% RSLogix 500 project Unscrambler_D.RSS, saved by version 12.00.00.00 %
PROJECT "3234"    % processor: MicroLogix 1400 %

PROGRAM FILES
  LAD 2   15 rungs
  LAD 3   13 rungs
  LAD 4   2 rungs
  LAD 5   18 rungs
  LAD 6   37 rungs
  LAD 7   31 rungs
  LAD 8   105 rungs
  LAD 9, 10, 11, 12, 13, 14, 15: only END

DATA FILES
  O0 OUTPUT  6 elements
  I1 INPUT  9 elements
  S2 STATUS  66 elements
  B3 BINARY  32 elements
  T4 TIMER  40 elements
  C5 COUNTER  32 elements
  R6 CONTROL  16 elements
  N7 INTEGER  105 elements
  F8 FLOAT  1 elements
  N10   10 elements
  MG11   40 elements
  N12   2 elements
  N13   10 elements
  N17   1 elements
  ST23   32 elements
  N24   17 elements
  B27   1 elements

LADDER 2
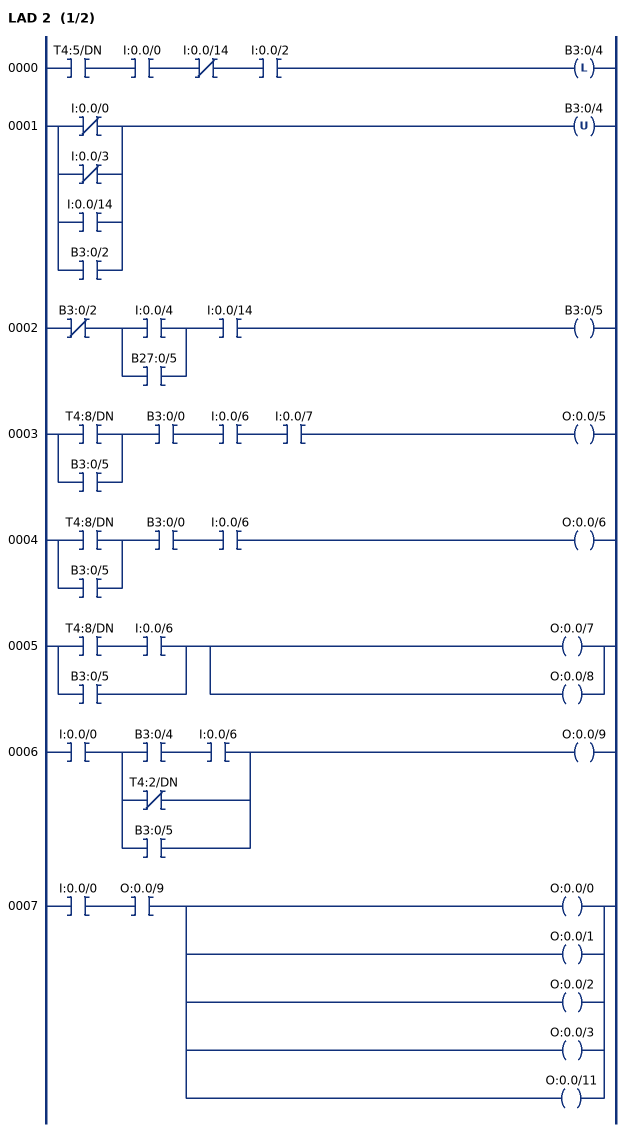
% Rung: 0 %
SOR XIC T4:5/DN XIC I:0.0/0 XIO I:0.0/14 XIC I:0.0/2 OTL B3:0/4 EOR
% Rung: 1 %
SOR BST XIO I:0.0/0 NXB XIO I:0.0/3 NXB XIC I:0.0/14 NXB XIC B3:0/2 BND OTU B3:0/4 EOR
% Rung: 2 %
SOR XIO B3:0/2 BST XIC I:0.0/4 NXB XIC B27:0/5 BND XIC I:0.0/14 OTE B3:0/5 EOR
% Rung: 3 %
SOR BST XIC T4:8/DN NXB XIC B3:0/5 BND XIC B3:0/0 XIC I:0.0/6 XIC I:0.0/7 OTE O:0.0/5 EOR
% Rung: 4 %
SOR BST XIC T4:8/DN NXB XIC B3:0/5 BND XIC B3:0/0 XIC I:0.0/6 OTE O:0.0/6 EOR
% Rung: 5 %
SOR BST XIC T4:8/DN XIC I:0.0/6 NXB XIC B3:0/5 BND BST OTE O:0.0/7 NXB OTE O:0.0/8 BND EOR
% Rung: 6 %
SOR XIC I:0.0/0 BST XIC B3:0/4 XIC I:0.0/6 NXB XIO T4:2/DN NXB XIC B3:0/5 BND OTE O:0.0/9 EOR
% Rung: 7 %
SOR XIC I:0.0/0 XIC O:0.0/9 BST OTE O:0.0/0 NXB OTE O:0.0/1 NXB OTE O:0.0/2 NXB OTE O:0.0/3 NXB OTE O:0.0/11 BND EOR

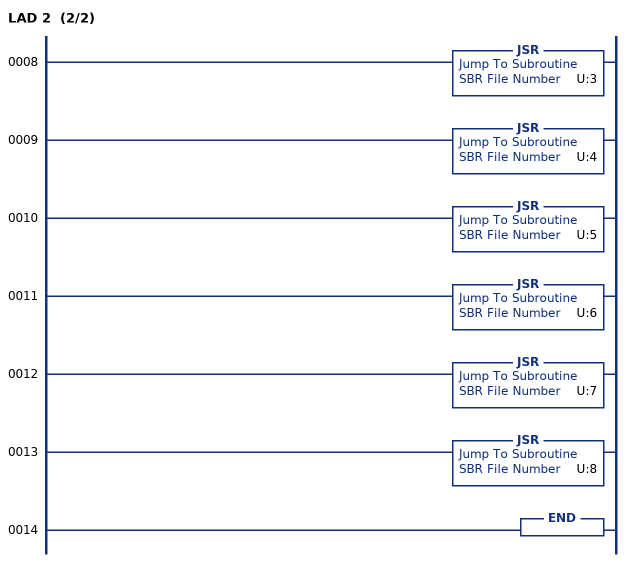
% Rung: 8 %
SOR JSR U:3 EOR
% Rung: 9 %
SOR JSR U:4 EOR
% Rung: 10 %
SOR JSR U:5 EOR
% Rung: 11 %
SOR JSR U:6 EOR
% Rung: 12 %
SOR JSR U:7 EOR
% Rung: 13 %
SOR JSR U:8 EOR
% Rung: 14 %
SOR END EOR

LADDER 3
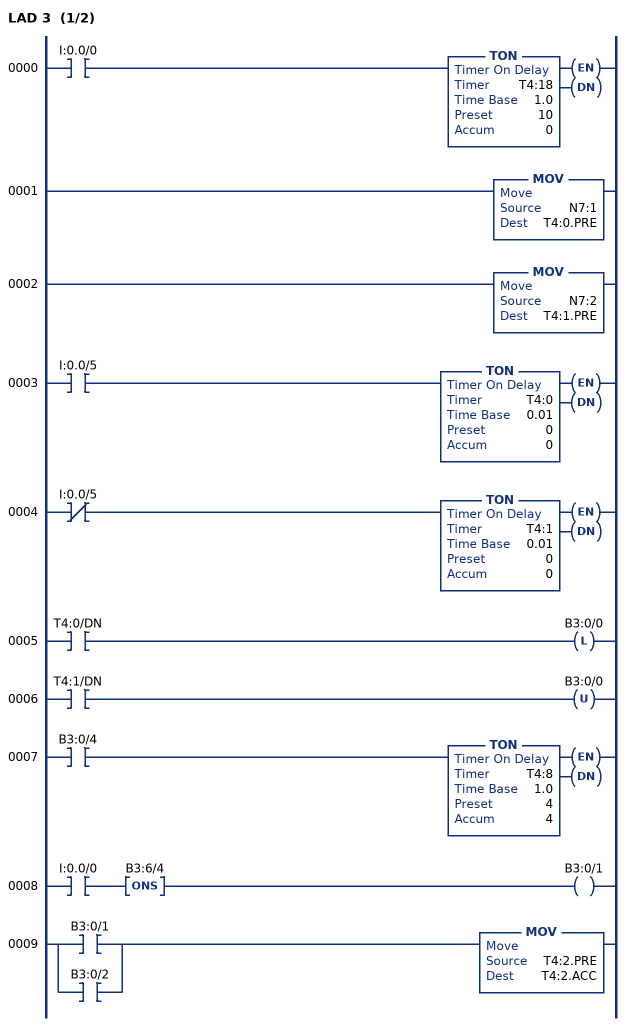
% Rung: 0 %
SOR XIC I:0.0/0 TON T4:18 1.0 10 0 EOR
% Rung: 1 %
SOR MOV N7:1 T4:0.PRE EOR
% Rung: 2 %
SOR MOV N7:2 T4:1.PRE EOR
% Rung: 3 %
SOR XIC I:0.0/5 TON T4:0 0.01 0 0 EOR
% Rung: 4 %
SOR XIO I:0.0/5 TON T4:1 0.01 0 0 EOR
% Rung: 5 %
SOR XIC T4:0/DN OTL B3:0/0 EOR
% Rung: 6 %
SOR XIC T4:1/DN OTU B3:0/0 EOR
% Rung: 7 %
SOR XIC B3:0/4 TON T4:8 1.0 4 4 EOR
% Rung: 8 %
SOR XIC I:0.0/0 ONS B3:6/4 OTE B3:0/1 EOR
% Rung: 9 %
SOR BST XIC B3:0/1 NXB XIC B3:0/2 BND MOV T4:2.PRE T4:2.ACC EOR

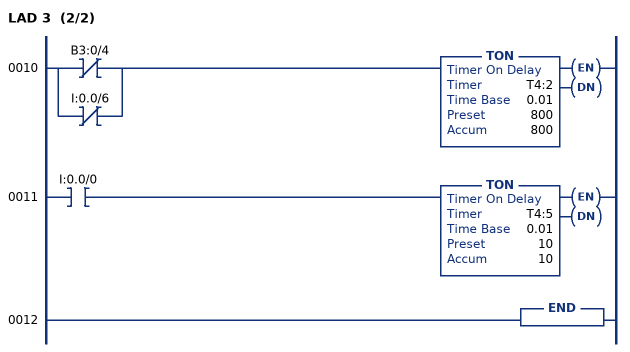
% Rung: 10 %
SOR BST XIO B3:0/4 NXB XIO I:0.0/6 BND TON T4:2 0.01 800 800 EOR
% Rung: 11 %
SOR XIC I:0.0/0 TON T4:5 0.01 10 10 EOR
% Rung: 12 %
SOR END EOR

LADDER 4
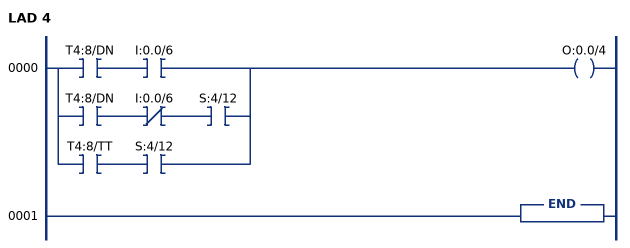
% Rung: 0 %
SOR BST XIC T4:8/DN XIC I:0.0/6 NXB XIC T4:8/DN XIO I:0.0/6 XIC S:4/12 NXB XIC T4:8/TT XIC S:4/12 BND OTE O:0.0/4 EOR
% Rung: 1 %
SOR END EOR

LADDER 5
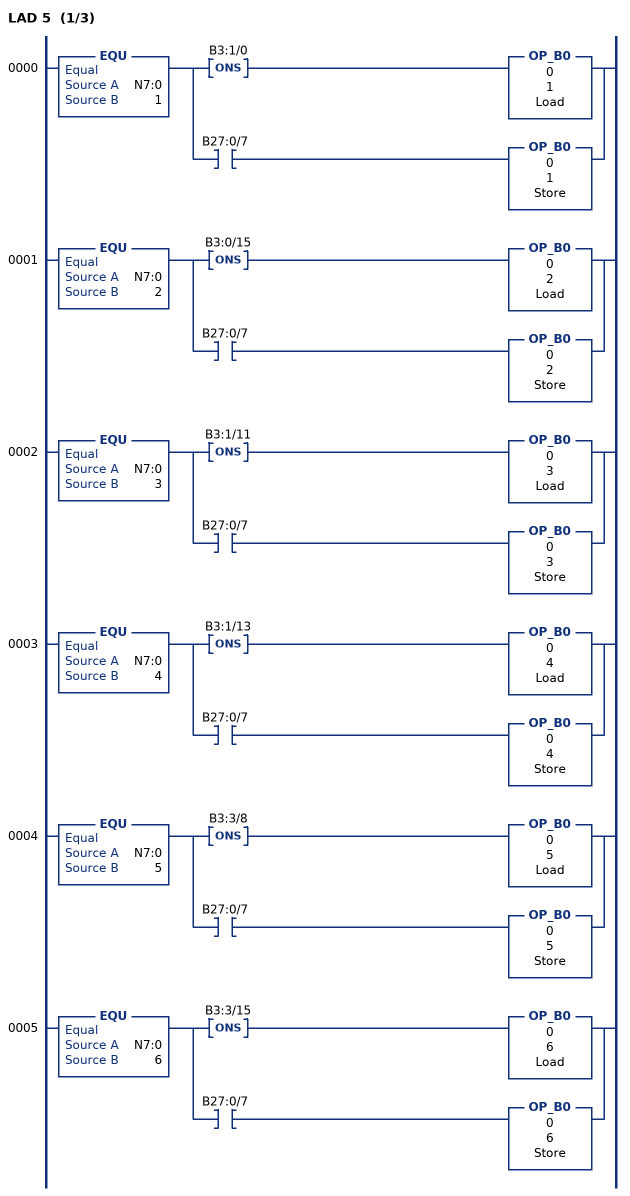
% Rung: 0 %
SOR EQU N7:0 1 BST ONS B3:1/0 OP_B0 0 1 Load NXB XIC B27:0/7 OP_B0 0 1 Store BND EOR
% Rung: 1 %
SOR EQU N7:0 2 BST ONS B3:0/15 OP_B0 0 2 Load NXB XIC B27:0/7 OP_B0 0 2 Store BND EOR
% Rung: 2 %
SOR EQU N7:0 3 BST ONS B3:1/11 OP_B0 0 3 Load NXB XIC B27:0/7 OP_B0 0 3 Store BND EOR
% Rung: 3 %
SOR EQU N7:0 4 BST ONS B3:1/13 OP_B0 0 4 Load NXB XIC B27:0/7 OP_B0 0 4 Store BND EOR
% Rung: 4 %
SOR EQU N7:0 5 BST ONS B3:3/8 OP_B0 0 5 Load NXB XIC B27:0/7 OP_B0 0 5 Store BND EOR
% Rung: 5 %
SOR EQU N7:0 6 BST ONS B3:3/15 OP_B0 0 6 Load NXB XIC B27:0/7 OP_B0 0 6 Store BND EOR

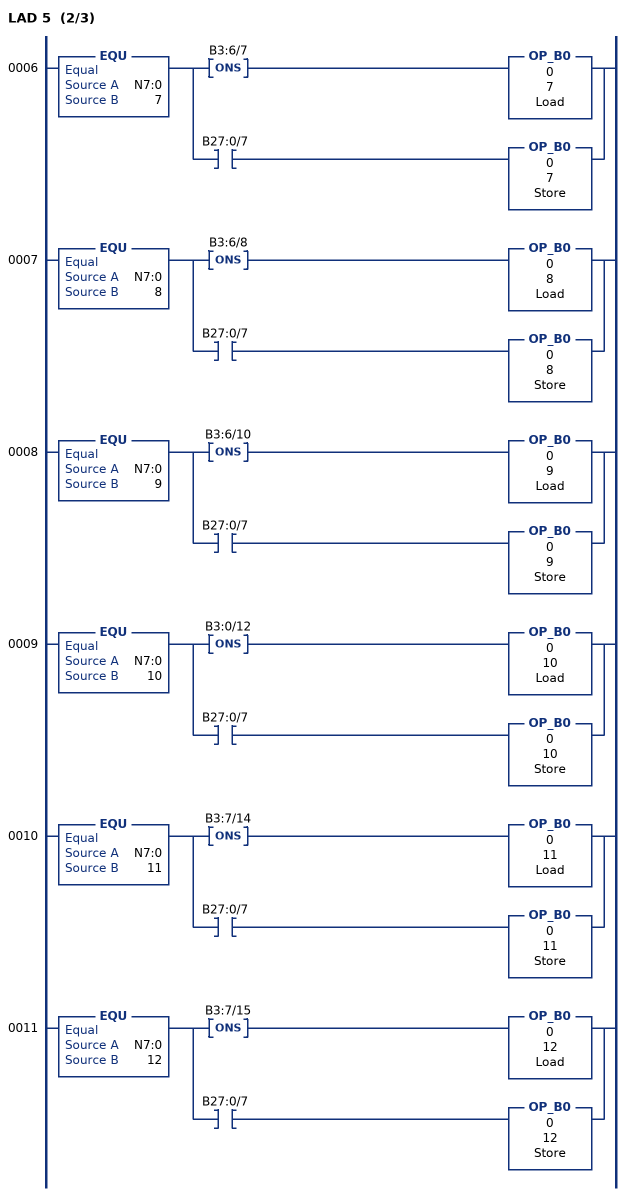
% Rung: 6 %
SOR EQU N7:0 7 BST ONS B3:6/7 OP_B0 0 7 Load NXB XIC B27:0/7 OP_B0 0 7 Store BND EOR
% Rung: 7 %
SOR EQU N7:0 8 BST ONS B3:6/8 OP_B0 0 8 Load NXB XIC B27:0/7 OP_B0 0 8 Store BND EOR
% Rung: 8 %
SOR EQU N7:0 9 BST ONS B3:6/10 OP_B0 0 9 Load NXB XIC B27:0/7 OP_B0 0 9 Store BND EOR
% Rung: 9 %
SOR EQU N7:0 10 BST ONS B3:0/12 OP_B0 0 10 Load NXB XIC B27:0/7 OP_B0 0 10 Store BND EOR
% Rung: 10 %
SOR EQU N7:0 11 BST ONS B3:7/14 OP_B0 0 11 Load NXB XIC B27:0/7 OP_B0 0 11 Store BND EOR
% Rung: 11 %
SOR EQU N7:0 12 BST ONS B3:7/15 OP_B0 0 12 Load NXB XIC B27:0/7 OP_B0 0 12 Store BND EOR

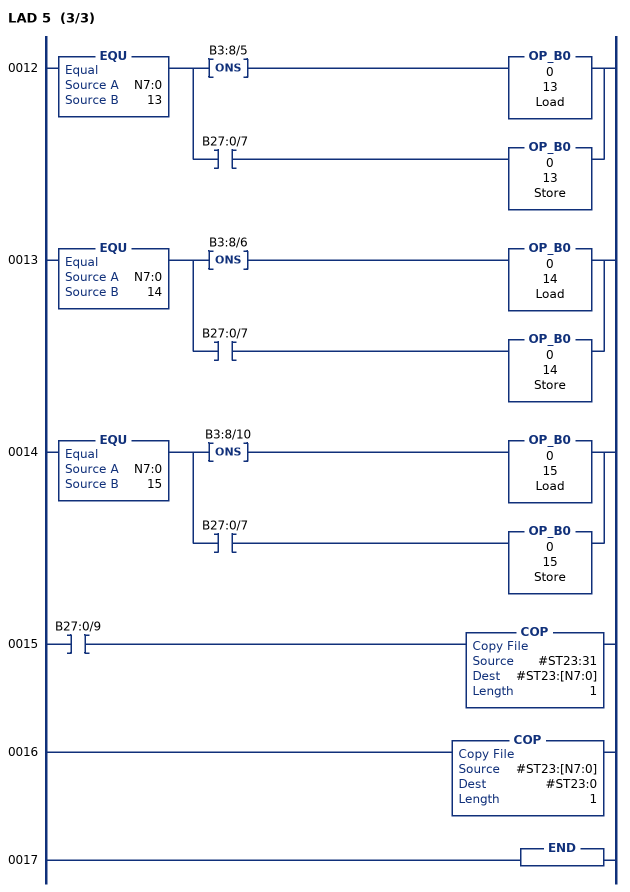
% Rung: 12 %
SOR EQU N7:0 13 BST ONS B3:8/5 OP_B0 0 13 Load NXB XIC B27:0/7 OP_B0 0 13 Store BND EOR
% Rung: 13 %
SOR EQU N7:0 14 BST ONS B3:8/6 OP_B0 0 14 Load NXB XIC B27:0/7 OP_B0 0 14 Store BND EOR
% Rung: 14 %
SOR EQU N7:0 15 BST ONS B3:8/10 OP_B0 0 15 Load NXB XIC B27:0/7 OP_B0 0 15 Store BND EOR
% Rung: 15 %
SOR XIC B27:0/9 COP #ST23:31 #ST23:[N7:0] 1 EOR
% Rung: 16 %
SOR COP #ST23:[N7:0] #ST23:0 1 EOR
% Rung: 17 %
SOR END EOR

LADDER 6
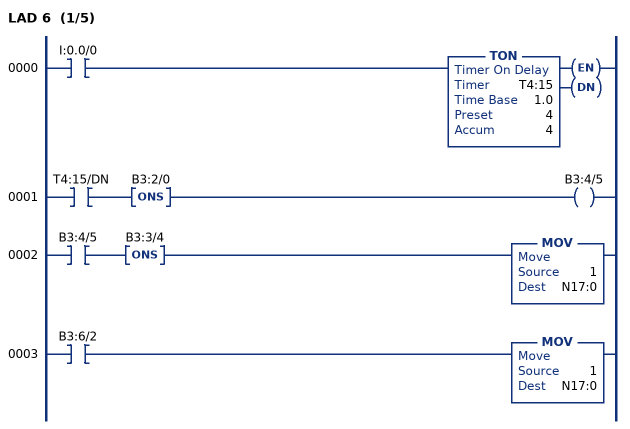
% Rung: 0 %
SOR XIC I:0.0/0 TON T4:15 1.0 4 4 EOR
% Rung: 1 %
SOR XIC T4:15/DN ONS B3:2/0 OTE B3:4/5 EOR
% Rung: 2 %
SOR XIC B3:4/5 ONS B3:3/4 MOV 1 N17:0 EOR
% Rung: 3 %
SOR XIC B3:6/2 MOV 1 N17:0 EOR

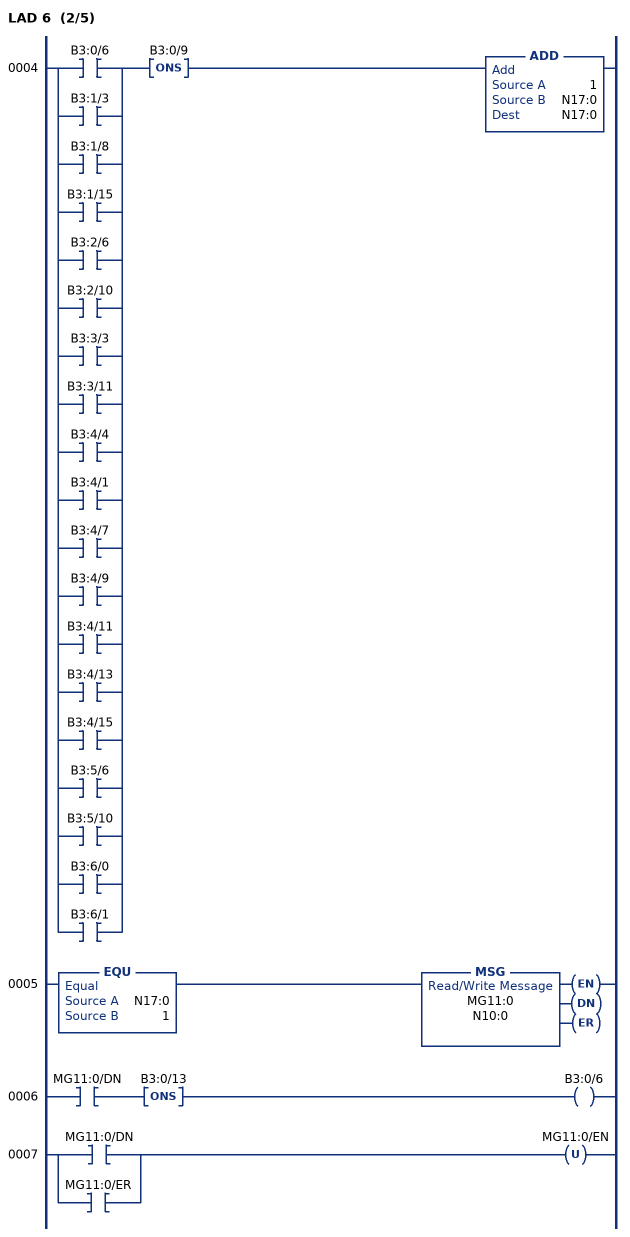
% Rung: 4 %
SOR BST XIC B3:0/6 NXB XIC B3:1/3 NXB XIC B3:1/8 NXB XIC B3:1/15 NXB XIC B3:2/6 NXB XIC B3:2/10 NXB XIC B3:3/3 NXB XIC B3:3/11 NXB XIC B3:4/4 NXB XIC B3:4/1 NXB XIC B3:4/7 NXB XIC B3:4/9 NXB XIC B3:4/11 NXB XIC B3:4/13 NXB XIC B3:4/15 NXB XIC B3:5/6 NXB XIC B3:5/10 NXB XIC B3:6/0 NXB XIC B3:6/1 BND ONS B3:0/9 ADD 1 N17:0 N17:0 EOR
% Rung: 5 %
SOR EQU N17:0 1 MSG MG11:0 N10:0 EOR
%   MSG set-up: 06 Write Single Register (4xxxxx) | 2 | 1 | 8194 | N10:0 | 0 | 1 | 0 | CLIENT              :502 | 0 | 0 | ? %
% Rung: 6 %
SOR XIC MG11:0/DN ONS B3:0/13 OTE B3:0/6 EOR
% Rung: 7 %
SOR BST XIC MG11:0/DN NXB XIC MG11:0/ER BND OTU MG11:0/EN EOR

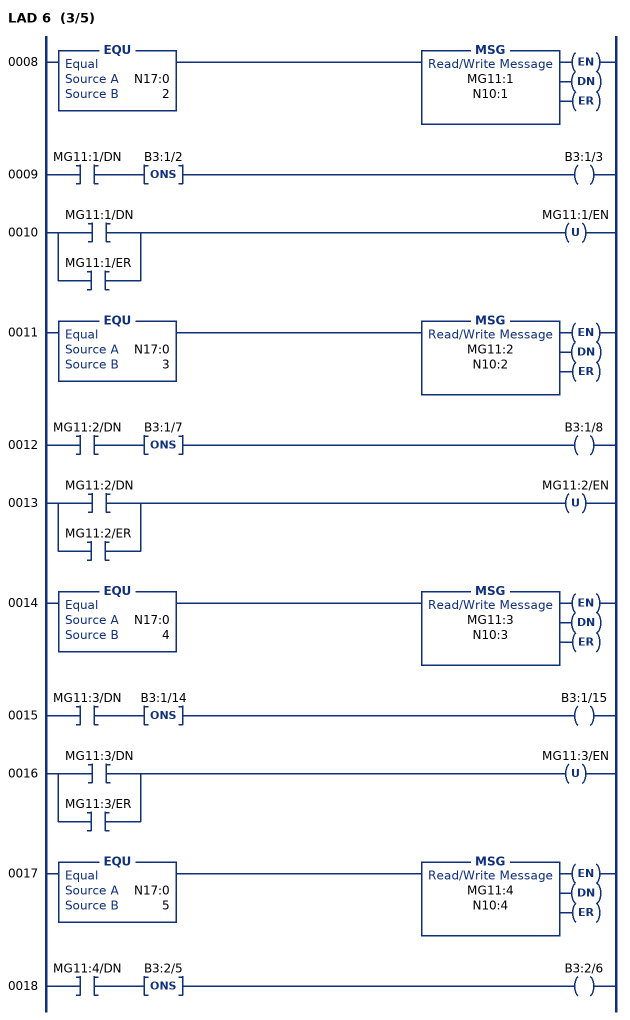
% Rung: 8 %
SOR EQU N17:0 2 MSG MG11:1 N10:1 EOR
%   MSG set-up: 06 Write Single Register (4xxxxx) | 2 | 1 | 8194 | N10:1 | 0 | 2 | 0 | CLIENT              :502 | 0 | 0 | ? %
% Rung: 9 %
SOR XIC MG11:1/DN ONS B3:1/2 OTE B3:1/3 EOR
% Rung: 10 %
SOR BST XIC MG11:1/DN NXB XIC MG11:1/ER BND OTU MG11:1/EN EOR
% Rung: 11 %
SOR EQU N17:0 3 MSG MG11:2 N10:2 EOR
%   MSG set-up: 06 Write Single Register (4xxxxx) | 2 | 1 | 8194 | N10:2 | 0 | 3 | 0 | CLIENT              :502 | 0 | 0 | ? %
% Rung: 12 %
SOR XIC MG11:2/DN ONS B3:1/7 OTE B3:1/8 EOR
% Rung: 13 %
SOR BST XIC MG11:2/DN NXB XIC MG11:2/ER BND OTU MG11:2/EN EOR
% Rung: 14 %
SOR EQU N17:0 4 MSG MG11:3 N10:3 EOR
%   MSG set-up: 06 Write Single Register (4xxxxx) | 2 | 1 | 8194 | N10:3 | 0 | 4 | 0 | CLIENT              :502 | 0 | 0 | ? %
% Rung: 15 %
SOR XIC MG11:3/DN ONS B3:1/14 OTE B3:1/15 EOR
% Rung: 16 %
SOR BST XIC MG11:3/DN NXB XIC MG11:3/ER BND OTU MG11:3/EN EOR
% Rung: 17 %
SOR EQU N17:0 5 MSG MG11:4 N10:4 EOR
%   MSG set-up: 06 Write Single Register (4xxxxx) | 2 | 1 | 8194 | N10:4 | 0 | 5 | 0 | CLIENT              :502 | 0 | 0 | ? %
% Rung: 18 %
SOR XIC MG11:4/DN ONS B3:2/5 OTE B3:2/6 EOR

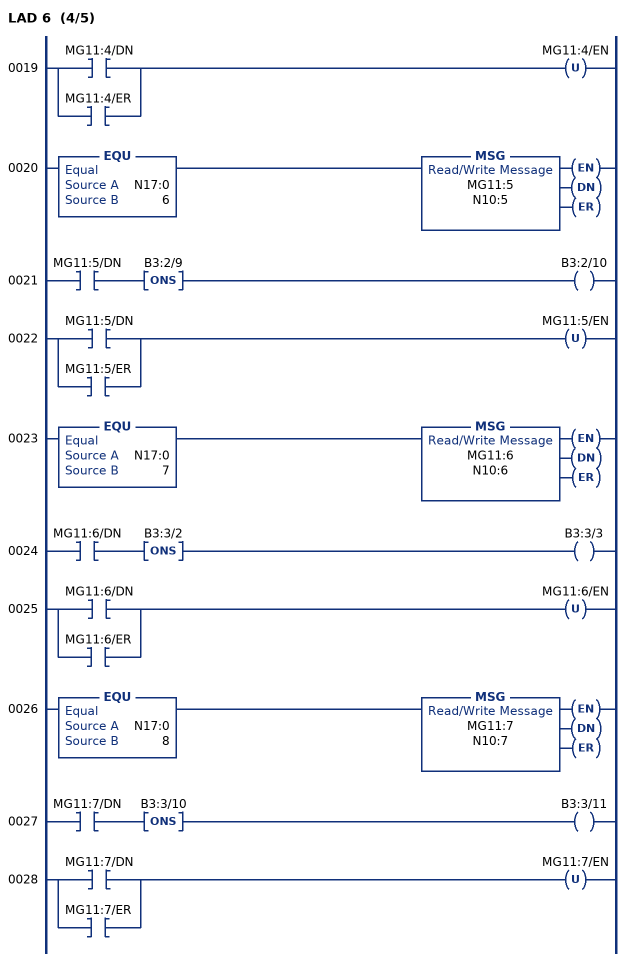
% Rung: 19 %
SOR BST XIC MG11:4/DN NXB XIC MG11:4/ER BND OTU MG11:4/EN EOR
% Rung: 20 %
SOR EQU N17:0 6 MSG MG11:5 N10:5 EOR
%   MSG set-up: 06 Write Single Register (4xxxxx) | 2 | 1 | 8194 | N10:5 | 0 | 6 | 0 | CLIENT              :502 | 0 | 0 | ? %
% Rung: 21 %
SOR XIC MG11:5/DN ONS B3:2/9 OTE B3:2/10 EOR
% Rung: 22 %
SOR BST XIC MG11:5/DN NXB XIC MG11:5/ER BND OTU MG11:5/EN EOR
% Rung: 23 %
SOR EQU N17:0 7 MSG MG11:6 N10:6 EOR
%   MSG set-up: 06 Write Single Register (4xxxxx) | 2 | 1 | 8194 | N10:6 | 0 | 7 | 0 | CLIENT              :502 | 0 | 0 | ? %
% Rung: 24 %
SOR XIC MG11:6/DN ONS B3:3/2 OTE B3:3/3 EOR
% Rung: 25 %
SOR BST XIC MG11:6/DN NXB XIC MG11:6/ER BND OTU MG11:6/EN EOR
% Rung: 26 %
SOR EQU N17:0 8 MSG MG11:7 N10:7 EOR
%   MSG set-up: 06 Write Single Register (4xxxxx) | 2 | 1 | 8194 | N10:7 | 0 | 8 | 0 | CLIENT              :502 | 0 | 0 | ? %
% Rung: 27 %
SOR XIC MG11:7/DN ONS B3:3/10 OTE B3:3/11 EOR
% Rung: 28 %
SOR BST XIC MG11:7/DN NXB XIC MG11:7/ER BND OTU MG11:7/EN EOR

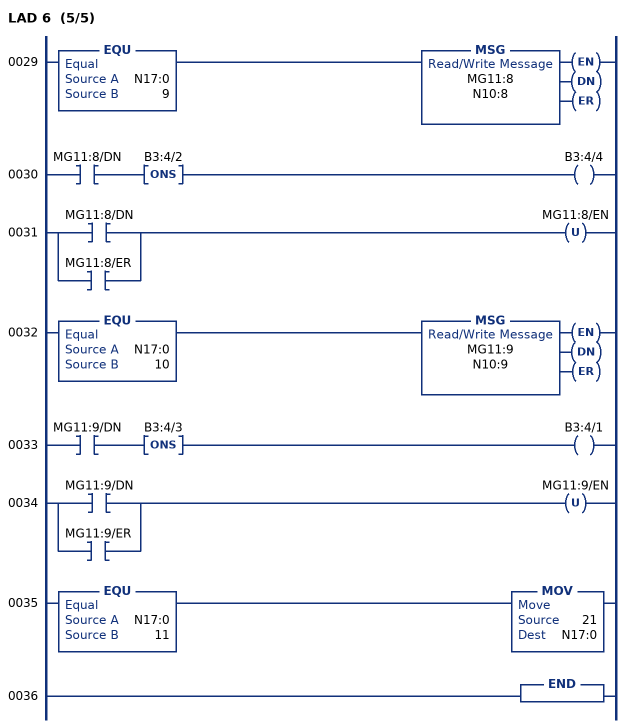
% Rung: 29 %
SOR EQU N17:0 9 MSG MG11:8 N10:8 EOR
%   MSG set-up: 06 Write Single Register (4xxxxx) | 2 | 1 | 8194 | N10:8 | 0 | 9 | 0 | CLIENT              :502 | 0 | 0 | ? %
% Rung: 30 %
SOR XIC MG11:8/DN ONS B3:4/2 OTE B3:4/4 EOR
% Rung: 31 %
SOR BST XIC MG11:8/DN NXB XIC MG11:8/ER BND OTU MG11:8/EN EOR
% Rung: 32 %
SOR EQU N17:0 10 MSG MG11:9 N10:9 EOR
%   MSG set-up: 06 Write Single Register (4xxxxx) | 2 | 1 | 8194 | N10:9 | 0 | 10 | 0 | CLIENT              :502 | 0 | 0 | ? %
% Rung: 33 %
SOR XIC MG11:9/DN ONS B3:4/3 OTE B3:4/1 EOR
% Rung: 34 %
SOR BST XIC MG11:9/DN NXB XIC MG11:9/ER BND OTU MG11:9/EN EOR
% Rung: 35 %
SOR EQU N17:0 11 MOV 21 N17:0 EOR
% Rung: 36 %
SOR END EOR

LADDER 7
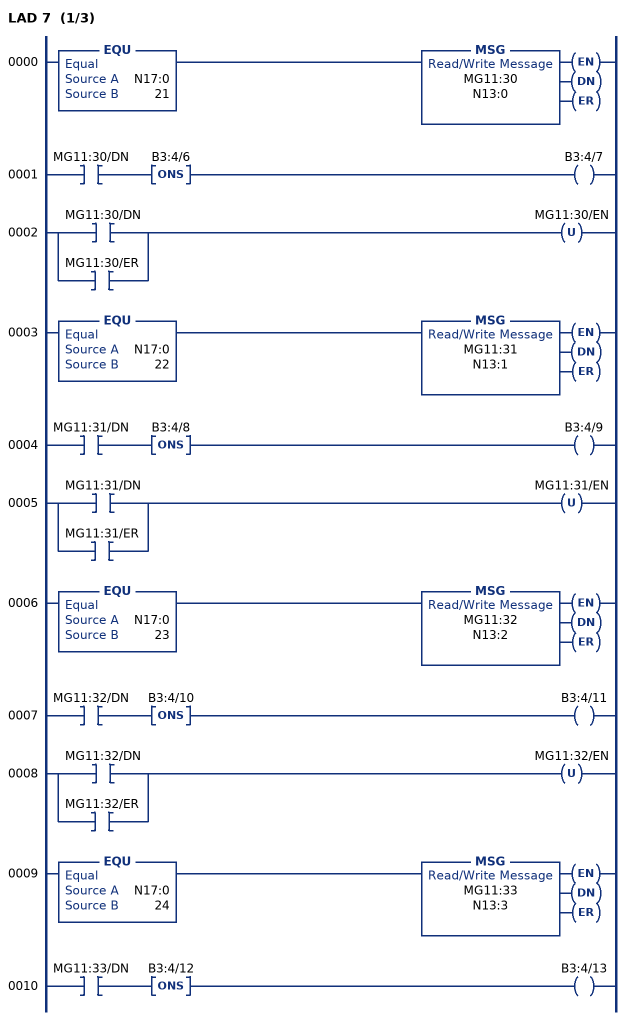
% Rung: 0 %
SOR EQU N17:0 21 MSG MG11:30 N13:0 EOR
%   MSG set-up: 03 Read Holding Registers (4xxxxx) | 5 | 1 | 8449 | N13:0 | 0 | 1 | 0 | CLIENT              :502 | 0 | 0 | ? %
% Rung: 1 %
SOR XIC MG11:30/DN ONS B3:4/6 OTE B3:4/7 EOR
% Rung: 2 %
SOR BST XIC MG11:30/DN NXB XIC MG11:30/ER BND OTU MG11:30/EN EOR
% Rung: 3 %
SOR EQU N17:0 22 MSG MG11:31 N13:1 EOR
%   MSG set-up: 03 Read Holding Registers (4xxxxx) | 5 | 1 | 8449 | N13:1 | 0 | 2 | 0 | CLIENT              :502 | 0 | 0 | ? %
% Rung: 4 %
SOR XIC MG11:31/DN ONS B3:4/8 OTE B3:4/9 EOR
% Rung: 5 %
SOR BST XIC MG11:31/DN NXB XIC MG11:31/ER BND OTU MG11:31/EN EOR
% Rung: 6 %
SOR EQU N17:0 23 MSG MG11:32 N13:2 EOR
%   MSG set-up: 03 Read Holding Registers (4xxxxx) | 5 | 1 | 8449 | N13:2 | 0 | 3 | 0 | CLIENT              :502 | 0 | 0 | ? %
% Rung: 7 %
SOR XIC MG11:32/DN ONS B3:4/10 OTE B3:4/11 EOR
% Rung: 8 %
SOR BST XIC MG11:32/DN NXB XIC MG11:32/ER BND OTU MG11:32/EN EOR
% Rung: 9 %
SOR EQU N17:0 24 MSG MG11:33 N13:3 EOR
%   MSG set-up: 03 Read Holding Registers (4xxxxx) | 5 | 1 | 8449 | N13:3 | 0 | 4 | 0 | CLIENT              :502 | 0 | 0 | ? %
% Rung: 10 %
SOR XIC MG11:33/DN ONS B3:4/12 OTE B3:4/13 EOR

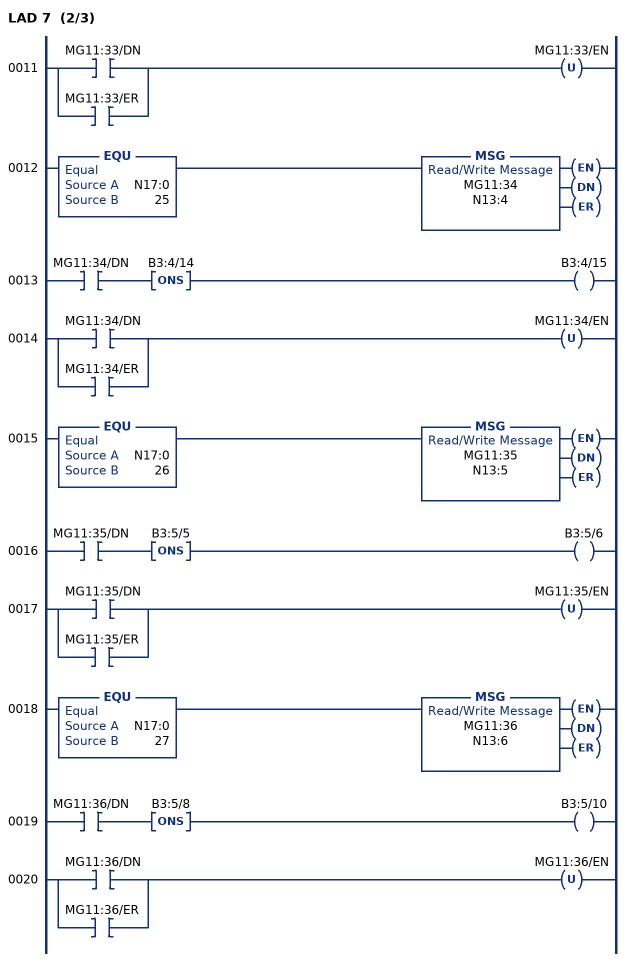
% Rung: 11 %
SOR BST XIC MG11:33/DN NXB XIC MG11:33/ER BND OTU MG11:33/EN EOR
% Rung: 12 %
SOR EQU N17:0 25 MSG MG11:34 N13:4 EOR
%   MSG set-up: 03 Read Holding Registers (4xxxxx) | 5 | 1 | 8449 | N13:4 | 0 | 5 | 0 | CLIENT              :502 | 0 | 0 | ? %
% Rung: 13 %
SOR XIC MG11:34/DN ONS B3:4/14 OTE B3:4/15 EOR
% Rung: 14 %
SOR BST XIC MG11:34/DN NXB XIC MG11:34/ER BND OTU MG11:34/EN EOR
% Rung: 15 %
SOR EQU N17:0 26 MSG MG11:35 N13:5 EOR
%   MSG set-up: 03 Read Holding Registers (4xxxxx) | 5 | 1 | 8449 | N13:5 | 0 | 6 | 0 | CLIENT              :502 | 0 | 0 | ? %
% Rung: 16 %
SOR XIC MG11:35/DN ONS B3:5/5 OTE B3:5/6 EOR
% Rung: 17 %
SOR BST XIC MG11:35/DN NXB XIC MG11:35/ER BND OTU MG11:35/EN EOR
% Rung: 18 %
SOR EQU N17:0 27 MSG MG11:36 N13:6 EOR
%   MSG set-up: 03 Read Holding Registers (4xxxxx) | 5 | 1 | 8449 | N13:6 | 0 | 7 | 0 | CLIENT              :502 | 0 | 0 | ? %
% Rung: 19 %
SOR XIC MG11:36/DN ONS B3:5/8 OTE B3:5/10 EOR
% Rung: 20 %
SOR BST XIC MG11:36/DN NXB XIC MG11:36/ER BND OTU MG11:36/EN EOR

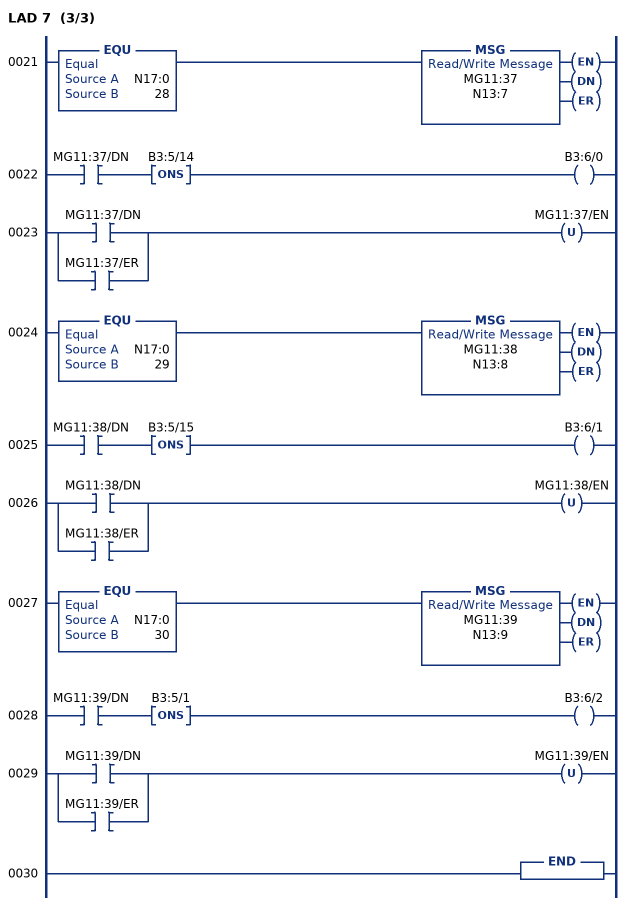
% Rung: 21 %
SOR EQU N17:0 28 MSG MG11:37 N13:7 EOR
%   MSG set-up: 03 Read Holding Registers (4xxxxx) | 5 | 1 | 8449 | N13:7 | 0 | 8 | 0 | CLIENT              :502 | 0 | 0 | ? %
% Rung: 22 %
SOR XIC MG11:37/DN ONS B3:5/14 OTE B3:6/0 EOR
% Rung: 23 %
SOR BST XIC MG11:37/DN NXB XIC MG11:37/ER BND OTU MG11:37/EN EOR
% Rung: 24 %
SOR EQU N17:0 29 MSG MG11:38 N13:8 EOR
%   MSG set-up: 03 Read Holding Registers (4xxxxx) | 5 | 1 | 8449 | N13:8 | 0 | 9 | 0 | CLIENT              :502 | 0 | 0 | ? %
% Rung: 25 %
SOR XIC MG11:38/DN ONS B3:5/15 OTE B3:6/1 EOR
% Rung: 26 %
SOR BST XIC MG11:38/DN NXB XIC MG11:38/ER BND OTU MG11:38/EN EOR
% Rung: 27 %
SOR EQU N17:0 30 MSG MG11:39 N13:9 EOR
%   MSG set-up: 03 Read Holding Registers (4xxxxx) | 5 | 1 | 8449 | N13:9 | 0 | 10 | 0 | CLIENT              :502 | 0 | 0 | ? %
% Rung: 28 %
SOR XIC MG11:39/DN ONS B3:5/1 OTE B3:6/2 EOR
% Rung: 29 %
SOR BST XIC MG11:39/DN NXB XIC MG11:39/ER BND OTU MG11:39/EN EOR
% Rung: 30 %
SOR END EOR

LADDER 8
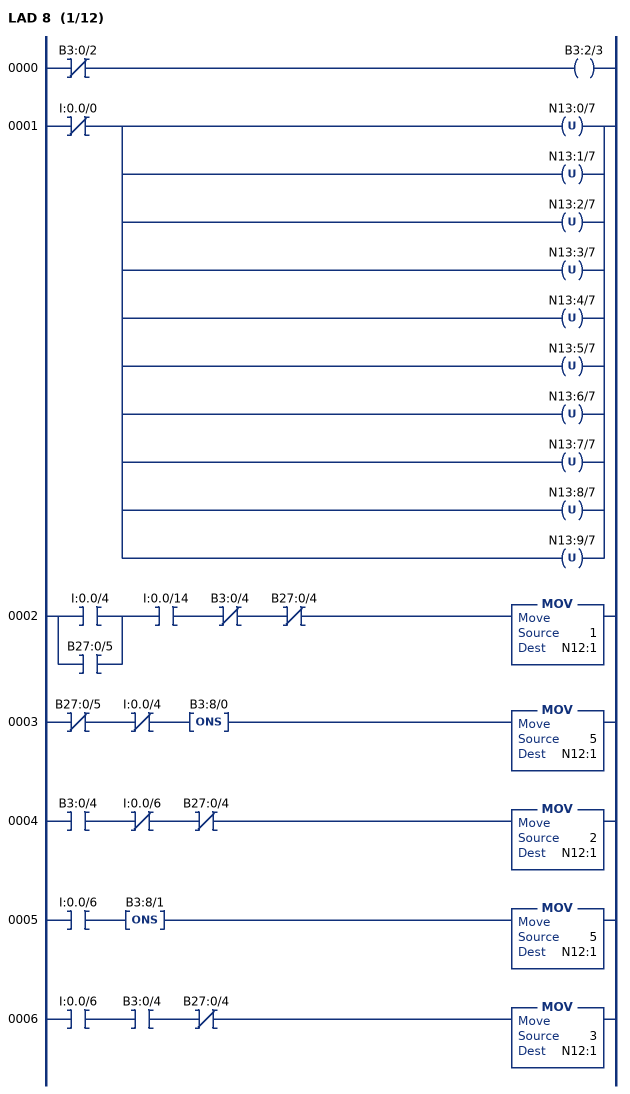
% Rung: 0 %
SOR XIO B3:0/2 OTE B3:2/3 EOR
% Rung: 1 %
SOR XIO I:0.0/0 BST OTU N13:0/7 NXB OTU N13:1/7 NXB OTU N13:2/7 NXB OTU N13:3/7 NXB OTU N13:4/7 NXB OTU N13:5/7 NXB OTU N13:6/7 NXB OTU N13:7/7 NXB OTU N13:8/7 NXB OTU N13:9/7 BND EOR
% Rung: 2 %
SOR BST XIC I:0.0/4 NXB XIC B27:0/5 BND XIC I:0.0/14 XIO B3:0/4 XIO B27:0/4 MOV 1 N12:1 EOR
% Rung: 3 %
SOR XIO B27:0/5 XIO I:0.0/4 ONS B3:8/0 MOV 5 N12:1 EOR
% Rung: 4 %
SOR XIC B3:0/4 XIO I:0.0/6 XIO B27:0/4 MOV 2 N12:1 EOR
% Rung: 5 %
SOR XIC I:0.0/6 ONS B3:8/1 MOV 5 N12:1 EOR
% Rung: 6 %
SOR XIC I:0.0/6 XIC B3:0/4 XIO B27:0/4 MOV 3 N12:1 EOR

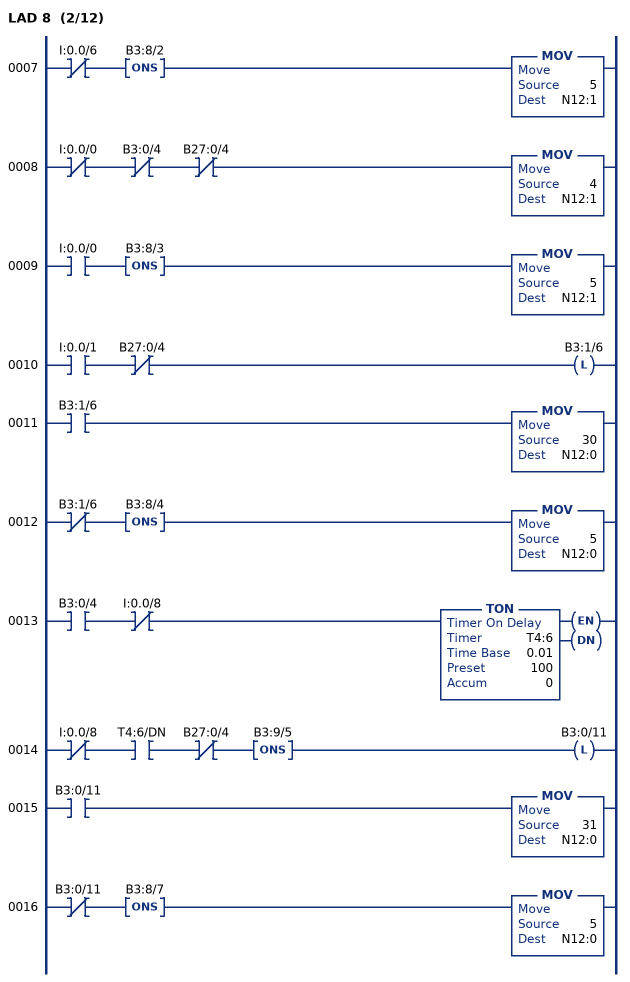
% Rung: 7 %
SOR XIO I:0.0/6 ONS B3:8/2 MOV 5 N12:1 EOR
% Rung: 8 %
SOR XIO I:0.0/0 XIO B3:0/4 XIO B27:0/4 MOV 4 N12:1 EOR
% Rung: 9 %
SOR XIC I:0.0/0 ONS B3:8/3 MOV 5 N12:1 EOR
% Rung: 10 %
SOR XIC I:0.0/1 XIO B27:0/4 OTL B3:1/6 EOR
% Rung: 11 %
SOR XIC B3:1/6 MOV 30 N12:0 EOR
% Rung: 12 %
SOR XIO B3:1/6 ONS B3:8/4 MOV 5 N12:0 EOR
% Rung: 13 %
SOR XIC B3:0/4 XIO I:0.0/8 TON T4:6 0.01 100 0 EOR
% Rung: 14 %
SOR XIO I:0.0/8 XIC T4:6/DN XIO B27:0/4 ONS B3:9/5 OTL B3:0/11 EOR
% Rung: 15 %
SOR XIC B3:0/11 MOV 31 N12:0 EOR
% Rung: 16 %
SOR XIO B3:0/11 ONS B3:8/7 MOV 5 N12:0 EOR

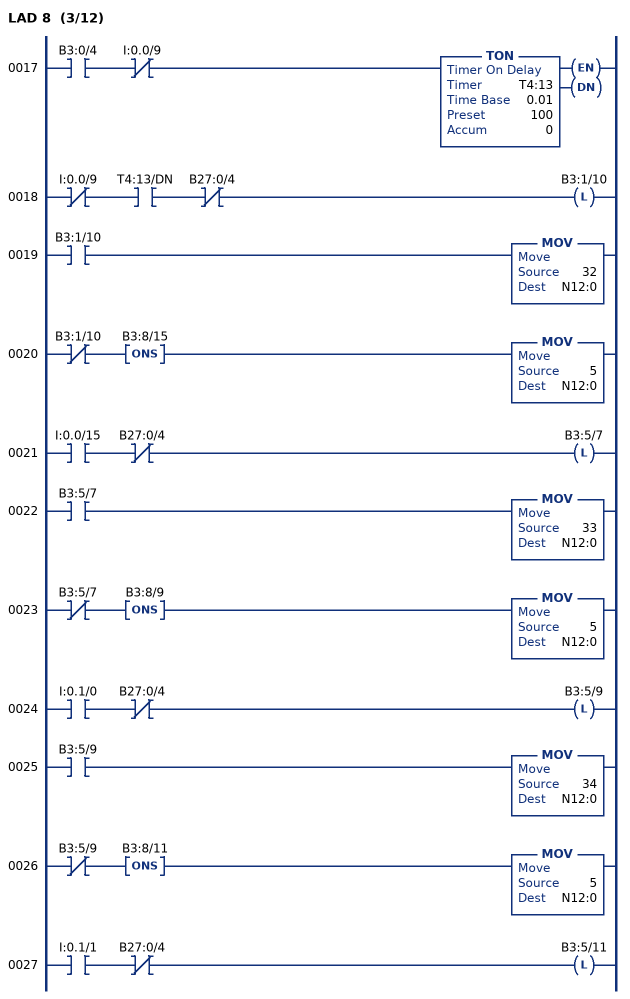
% Rung: 17 %
SOR XIC B3:0/4 XIO I:0.0/9 TON T4:13 0.01 100 0 EOR
% Rung: 18 %
SOR XIO I:0.0/9 XIC T4:13/DN XIO B27:0/4 OTL B3:1/10 EOR
% Rung: 19 %
SOR XIC B3:1/10 MOV 32 N12:0 EOR
% Rung: 20 %
SOR XIO B3:1/10 ONS B3:8/15 MOV 5 N12:0 EOR
% Rung: 21 %
SOR XIC I:0.0/15 XIO B27:0/4 OTL B3:5/7 EOR
% Rung: 22 %
SOR XIC B3:5/7 MOV 33 N12:0 EOR
% Rung: 23 %
SOR XIO B3:5/7 ONS B3:8/9 MOV 5 N12:0 EOR
% Rung: 24 %
SOR XIC I:0.1/0 XIO B27:0/4 OTL B3:5/9 EOR
% Rung: 25 %
SOR XIC B3:5/9 MOV 34 N12:0 EOR
% Rung: 26 %
SOR XIO B3:5/9 ONS B3:8/11 MOV 5 N12:0 EOR
% Rung: 27 %
SOR XIC I:0.1/1 XIO B27:0/4 OTL B3:5/11 EOR

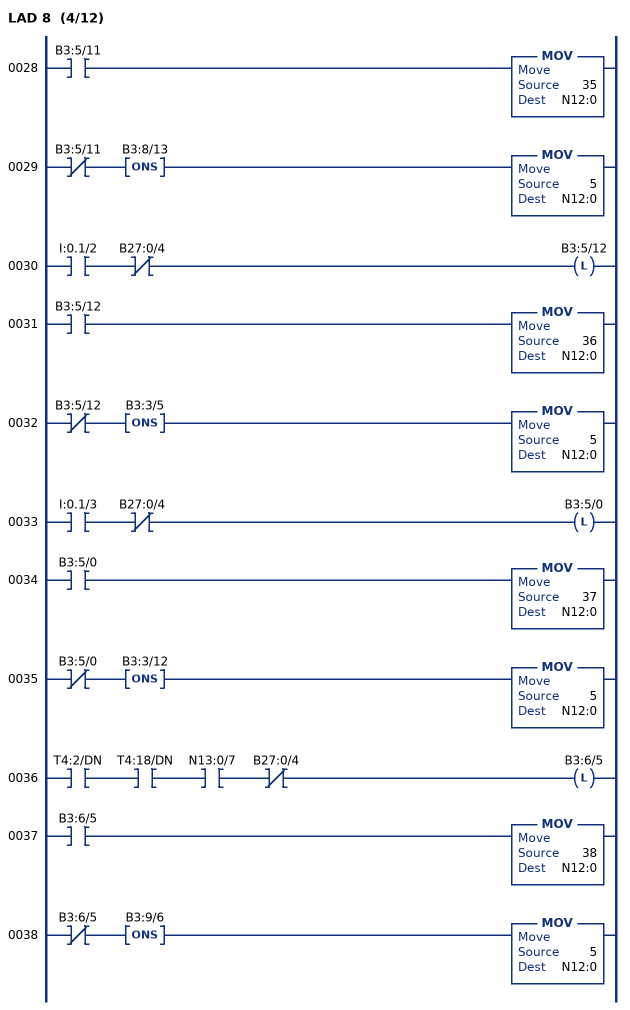
% Rung: 28 %
SOR XIC B3:5/11 MOV 35 N12:0 EOR
% Rung: 29 %
SOR XIO B3:5/11 ONS B3:8/13 MOV 5 N12:0 EOR
% Rung: 30 %
SOR XIC I:0.1/2 XIO B27:0/4 OTL B3:5/12 EOR
% Rung: 31 %
SOR XIC B3:5/12 MOV 36 N12:0 EOR
% Rung: 32 %
SOR XIO B3:5/12 ONS B3:3/5 MOV 5 N12:0 EOR
% Rung: 33 %
SOR XIC I:0.1/3 XIO B27:0/4 OTL B3:5/0 EOR
% Rung: 34 %
SOR XIC B3:5/0 MOV 37 N12:0 EOR
% Rung: 35 %
SOR XIO B3:5/0 ONS B3:3/12 MOV 5 N12:0 EOR
% Rung: 36 %
SOR XIC T4:2/DN XIC T4:18/DN XIC N13:0/7 XIO B27:0/4 OTL B3:6/5 EOR
% Rung: 37 %
SOR XIC B3:6/5 MOV 38 N12:0 EOR
% Rung: 38 %
SOR XIO B3:6/5 ONS B3:9/6 MOV 5 N12:0 EOR

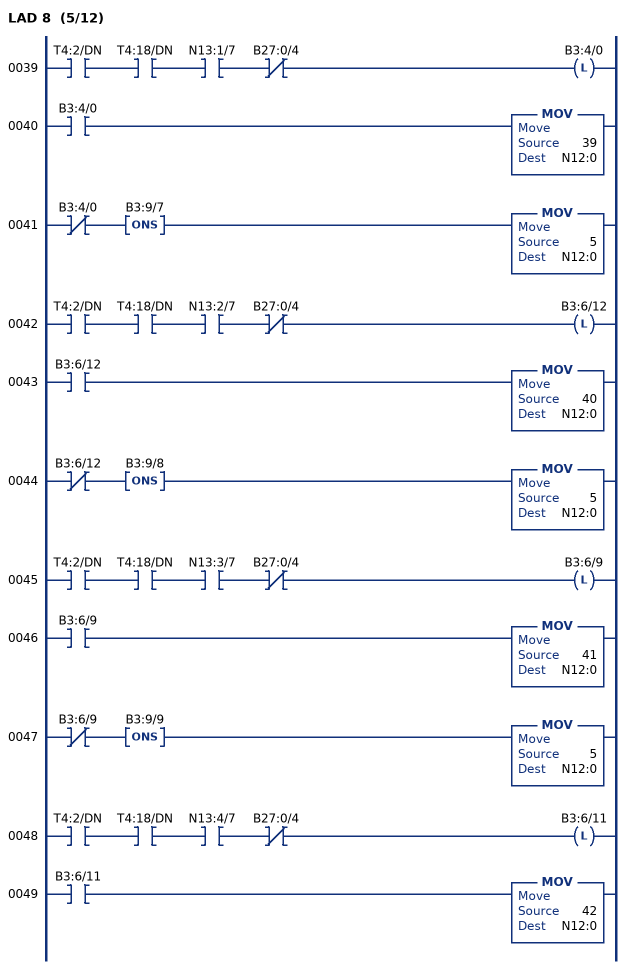
% Rung: 39 %
SOR XIC T4:2/DN XIC T4:18/DN XIC N13:1/7 XIO B27:0/4 OTL B3:4/0 EOR
% Rung: 40 %
SOR XIC B3:4/0 MOV 39 N12:0 EOR
% Rung: 41 %
SOR XIO B3:4/0 ONS B3:9/7 MOV 5 N12:0 EOR
% Rung: 42 %
SOR XIC T4:2/DN XIC T4:18/DN XIC N13:2/7 XIO B27:0/4 OTL B3:6/12 EOR
% Rung: 43 %
SOR XIC B3:6/12 MOV 40 N12:0 EOR
% Rung: 44 %
SOR XIO B3:6/12 ONS B3:9/8 MOV 5 N12:0 EOR
% Rung: 45 %
SOR XIC T4:2/DN XIC T4:18/DN XIC N13:3/7 XIO B27:0/4 OTL B3:6/9 EOR
% Rung: 46 %
SOR XIC B3:6/9 MOV 41 N12:0 EOR
% Rung: 47 %
SOR XIO B3:6/9 ONS B3:9/9 MOV 5 N12:0 EOR
% Rung: 48 %
SOR XIC T4:2/DN XIC T4:18/DN XIC N13:4/7 XIO B27:0/4 OTL B3:6/11 EOR
% Rung: 49 %
SOR XIC B3:6/11 MOV 42 N12:0 EOR

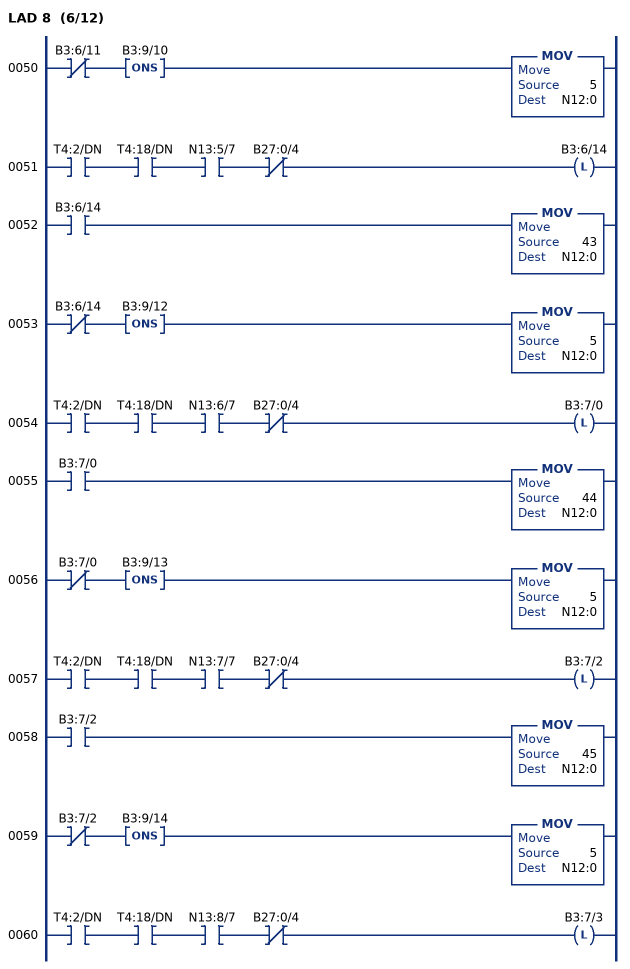
% Rung: 50 %
SOR XIO B3:6/11 ONS B3:9/10 MOV 5 N12:0 EOR
% Rung: 51 %
SOR XIC T4:2/DN XIC T4:18/DN XIC N13:5/7 XIO B27:0/4 OTL B3:6/14 EOR
% Rung: 52 %
SOR XIC B3:6/14 MOV 43 N12:0 EOR
% Rung: 53 %
SOR XIO B3:6/14 ONS B3:9/12 MOV 5 N12:0 EOR
% Rung: 54 %
SOR XIC T4:2/DN XIC T4:18/DN XIC N13:6/7 XIO B27:0/4 OTL B3:7/0 EOR
% Rung: 55 %
SOR XIC B3:7/0 MOV 44 N12:0 EOR
% Rung: 56 %
SOR XIO B3:7/0 ONS B3:9/13 MOV 5 N12:0 EOR
% Rung: 57 %
SOR XIC T4:2/DN XIC T4:18/DN XIC N13:7/7 XIO B27:0/4 OTL B3:7/2 EOR
% Rung: 58 %
SOR XIC B3:7/2 MOV 45 N12:0 EOR
% Rung: 59 %
SOR XIO B3:7/2 ONS B3:9/14 MOV 5 N12:0 EOR
% Rung: 60 %
SOR XIC T4:2/DN XIC T4:18/DN XIC N13:8/7 XIO B27:0/4 OTL B3:7/3 EOR

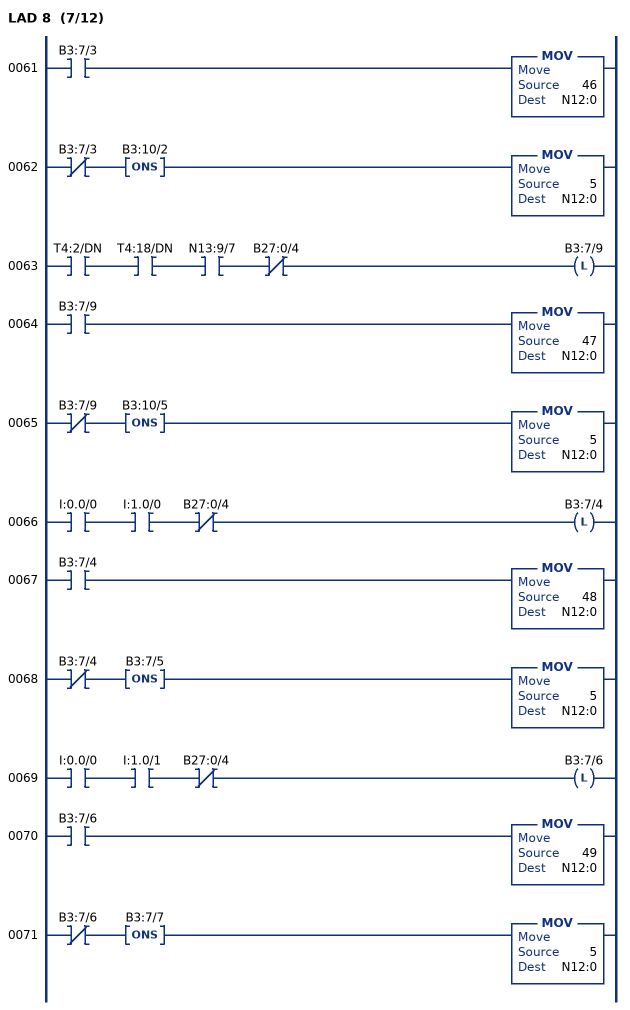
% Rung: 61 %
SOR XIC B3:7/3 MOV 46 N12:0 EOR
% Rung: 62 %
SOR XIO B3:7/3 ONS B3:10/2 MOV 5 N12:0 EOR
% Rung: 63 %
SOR XIC T4:2/DN XIC T4:18/DN XIC N13:9/7 XIO B27:0/4 OTL B3:7/9 EOR
% Rung: 64 %
SOR XIC B3:7/9 MOV 47 N12:0 EOR
% Rung: 65 %
SOR XIO B3:7/9 ONS B3:10/5 MOV 5 N12:0 EOR
% Rung: 66 %
SOR XIC I:0.0/0 XIC I:1.0/0 XIO B27:0/4 OTL B3:7/4 EOR
% Rung: 67 %
SOR XIC B3:7/4 MOV 48 N12:0 EOR
% Rung: 68 %
SOR XIO B3:7/4 ONS B3:7/5 MOV 5 N12:0 EOR
% Rung: 69 %
SOR XIC I:0.0/0 XIC I:1.0/1 XIO B27:0/4 OTL B3:7/6 EOR
% Rung: 70 %
SOR XIC B3:7/6 MOV 49 N12:0 EOR
% Rung: 71 %
SOR XIO B3:7/6 ONS B3:7/7 MOV 5 N12:0 EOR

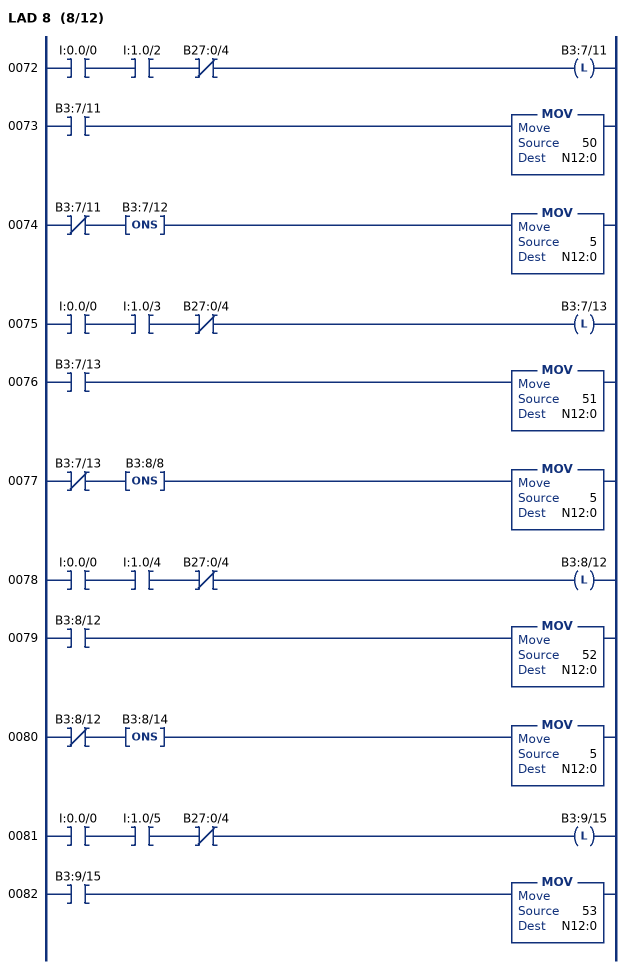
% Rung: 72 %
SOR XIC I:0.0/0 XIC I:1.0/2 XIO B27:0/4 OTL B3:7/11 EOR
% Rung: 73 %
SOR XIC B3:7/11 MOV 50 N12:0 EOR
% Rung: 74 %
SOR XIO B3:7/11 ONS B3:7/12 MOV 5 N12:0 EOR
% Rung: 75 %
SOR XIC I:0.0/0 XIC I:1.0/3 XIO B27:0/4 OTL B3:7/13 EOR
% Rung: 76 %
SOR XIC B3:7/13 MOV 51 N12:0 EOR
% Rung: 77 %
SOR XIO B3:7/13 ONS B3:8/8 MOV 5 N12:0 EOR
% Rung: 78 %
SOR XIC I:0.0/0 XIC I:1.0/4 XIO B27:0/4 OTL B3:8/12 EOR
% Rung: 79 %
SOR XIC B3:8/12 MOV 52 N12:0 EOR
% Rung: 80 %
SOR XIO B3:8/12 ONS B3:8/14 MOV 5 N12:0 EOR
% Rung: 81 %
SOR XIC I:0.0/0 XIC I:1.0/5 XIO B27:0/4 OTL B3:9/15 EOR
% Rung: 82 %
SOR XIC B3:9/15 MOV 53 N12:0 EOR

